FUNCTION_BLOCK TCPIP_Base
VAR_INPUT
END_VAR
VAR_OUTPUT
END_VAR
VAR
	connectToServer : SocketConnectTask;
	closeConectionToServer : SocketCloseTask;
	getReceivedDataFromServer : SocketRecieveTask;
	iState : INT;
	_connect: BOOL;
	_remoteIP : T_IPv4Addr;
	_remotePort : UDINT;
	_remoteHandle : Tc2_TcpIp.T_HSOCKET;
	clearRecieve: BOOL;
	_disconnect: BOOL;
END_VAR

CASE iState OF
	0: 
		IF _connect THEN
			_connect := false;
			iState := 10;
		END_IF
		
	10:
		IF connectToServer.Execute(RemoteIPAddress := _remoteIP, 
									RemotePortNumber := _remotePort) THEN
			iState := 20;
		END_IF
		
	20:
		_remoteHandle := connectToServer.RemoteSocket;
		getReceivedDataFromServer.RemoteSocket := _remoteHandle;
		IF connectToServer.Done AND _remoteHandle.handle <> 0 THEN
			iState := 30;
		END_IF
	
	30:
		IF getReceivedDataFromServer.Execute() THEN
			iState := 40;
		END_IF
		
	40:
		IF getReceivedDataFromServer.Done THEN
			IF _disconnect THEN
				_disconnect := FALSE;
				iState := 50;
			ELSE
				iState := 30;
			END_IF
			
		END_IF
	
	50:
		IF closeConectionToServer.Execute(remoteSocket := _remoteHandle) THEN
			iState := 60;
		END_IF
		
	60:
		IF closeConectionToServer.Done THEN
			iState := 0;
		END_IF
		
			
END_CASE

connectToServer();
closeConectionToServer();
getReceivedDataFromServer();

METHOD ConnectToRobot : BOOL
VAR_INPUT
END_VAR
ConnectToRobot := _connect := true;
END_METHOD

METHOD DisconnectFromRobot : BOOL
VAR_INPUT
END_VAR
DisconnectFromRobot := _disconnect := true;
END_METHOD

METHOD PUBLIC GetData : ARRAY[0..1439] OF byte
VAR_INPUT
END_VAR
GetData := getReceivedDataFromServer.rxBuffer;
END_METHOD

PROPERTY PUBLIC RemoteServerIP : T_IPv4Addr
GET
RemoteServerIP := _remoteIP;
END_GET
SET
_remoteIP := RemoteServerIP;
END_SET
END_PROPERTY

PROPERTY PUBLIC RemoteServerPort : udint
GET
RemoteServerPort := _remotePort;
END_GET
SET
_remotePort := RemoteServerPort;
END_SET
END_PROPERTY

END_FUNCTION_BLOCK

(* stored: Version 1.1.0.1, ProductVersion 3.1.4024.12
   POU TCPIP_Base: Id {c12d86ef-055b-43b4-be43-8e1aa454c4be}, SpecialFunc None
   Method ConnectToRobot: Id {7fdcc8ae-a489-4d24-bc39-9edbb54156ec}
   Method DisconnectFromRobot: Id {a119b9c1-e6f5-4d3d-82d9-faa466d74979}
   Method GetData: Id {c410b5d6-710e-4806-8307-1c4cdc1466b5}
   Property RemoteServerIP: Id {71d05534-e3f9-431e-a916-9a11849cd730}
   Get Get: Id {ed5b35f5-8938-4a22-b10f-9fe33676c004}
   Set Set: Id {42094b82-ccda-4bfe-9e6a-91df50bb377b}
   Property RemoteServerPort: Id {f38399ff-a7cc-477b-a3d9-2a242f0fe26c}
   Get Get: Id {0fbd444c-fffa-46d7-b665-e3ae9b72b4ca}
   Set Set: Id {9f5ec062-55bf-4d37-ae87-9998f342cc59} *)
